FUNCTION_BLOCK FB_UpdatesParams
VAR_INPUT
	stHMIparams	:	ST_HMI_Params;
END_VAR
VAR_OUTPUT
	stParams	:	ST_CSL_Params;
END_VAR
VAR
END_VAR

stParams 				:=	FC_thresholdsCalculation(stHMIParams := stHMIParams);

stParams.Threshold 		:=	stHMIParams.Threshold;

stParams.BlueVoltage	:=	stHMIparams.BlueVoltage;
stParams.RedVoltage		:=	stHMIparams.RedVoltage;
stParams.WhiteVoltage	:=	stHMIparams.WhiteVoltage;

stParams.BlueSlot 		:=	stHMIparams.BlueSlot;
stParams.RedSlot  		:=	stHMIparams.RedSlot;
stParams.WhiteSlot		:=	stHMIparams.WhiteSlot;

stParams.StepSlot1		:=	stHMIparams.StepSlot1;
stParams.StepSlot2		:=	stHMIparams.StepSlot2;
stParams.StepSlot3		:=	stHMIparams.StepSlot3;
stParams.StepNoSlot		:=	stHMIparams.StepNoSlot;

stParams.StepPerRev		:=	stHMIparams.StepPerRev;

END_FUNCTION_BLOCK

(* stored: Version 1.1.0.1, ProductVersion 3.1.4024.12
   POU FB_UpdatesParams: Id {64458d58-651d-42fb-9cce-1fcf177958b7}, SpecialFunc None *)
